(* Logix 5000 project; controller EWEB_SOCK_TCP_CLIENT_VER2_1 1756-L63 rev 15.4; software revision 15.02 *)

TASK MainTask (periodic, rate 5 ms, priority 10, watchdog 500 ms) : MainProgram

MODULES
   Local : 1756-L63 (ICP 5, rev 15.4)
END_MODULES

TYPE OpenConnParam :
STRUCT
   Timeout : DINT;
   DestAddr : STRING;
END_STRUCT
END_TYPE

TYPE READ_DATA_REQ :
STRUCT
   Timeout : DINT;
   BufLen : DINT;
END_STRUCT
END_TYPE

TYPE READ_RESP :
STRUCT
   FromAddr : SockAddr;
   READ_BUFF : STR_4096;
END_STRUCT
END_TYPE

TYPE REQUEST_PARAMETERS :
STRUCT
   Type : DINT;   // 1 - TCP 2- UPD
   Addr : SockAddr;
END_STRUCT
END_TYPE

TYPE SockAddr :
STRUCT
   Family : INT;   // Address Family Must be 2
   Port : INT;   // Port Number
   Addr : DINT;   // IP Address
END_STRUCT
END_TYPE

TYPE STR_4096 :
STRUCT
   LEN : DINT;
   DATA : SINT[4096];
END_STRUCT
END_TYPE

TYPE STR_480 :
STRUCT
   LEN : DINT;
   DATA : SINT[480];
END_STRUCT
END_TYPE

TYPE WRT_DATA :
STRUCT
   Timeout : DINT;
   ToAddr : SockAddr;
   Buffer : STR_480;
END_STRUCT
END_TYPE

VAR_GLOBAL   (* controller tags *)
   _EWEB_PATH : STRING := '$01$07';
   Accept : ALIAS FOR Log_Enable.2;
   Attrubute : ALIAS FOR Log_Enable.6;
   Buf_Len_Sent : DINT := 7;
   Change_Log_MSG : MESSAGE;
        MessageParameters(ServiceCode := 16#0010, LocalElement := Log_Enable, ...)
   CLOCK : DINT[7] := ([0] := 1998, [1] := 1, [2] := 7, [3] := 4, [4] := 26, [5] := 6, [6] := 739599);
   COLN : STRING := ':';
   Connect_MSG : MESSAGE;
        MessageParameters(ServiceCode := 16#004c, LocalElement := Sock_Open_Par, ...)
   Connect_Request : BOOL;   // Toggle This Bit to Connect to a Remote Server
   Create : ALIAS FOR Log_Enable.0;
   Create_Sock_MSG : MESSAGE;
        MessageParameters(ServiceCode := 16#004b, LocalElement := Socket, DestinationTag := Instance, ...)
   Create_Socket_Request : BOOL;   // Manually Toggle This Bit to Create Socket
   Del_All_Sockets_MSG : MESSAGE;
        MessageParameters(ServiceCode := 16#0051, ...)
   Delete : ALIAS FOR Log_Enable.5;
   Delete_All_Sockets_Request : BOOL;
   Delete_Socket_MSG : MESSAGE;
        MessageParameters(ServiceCode := 16#004f, ...)
   Delete_Socket_Request : BOOL;
   Dest_IP : STRING := '100.100.90.1';
   Dest_port : STRING := '?port=10001';
   Errors : ALIAS FOR Log_Enable.7;
   Get_Socket_Instance_MSG : MESSAGE;
        MessageParameters(ServiceCode := 16#0001, DestinationTag := Socket_Instance_DATA, ...)
   Get_Socket_Instance_Request : BOOL;
   Get_Socket_Object_MSG : MESSAGE;
        MessageParameters(ServiceCode := 16#0001, DestinationTag := Socket_Object_Class_Response, ...)
   Get_Socket_Object_Request : BOOL;
   HOUR : STRING := '4';
   Instance : DINT := 17538;
   Log_Enable : DINT;
   Log_old : DINT;
   MINUTE : STRING := '26';
   Nothing : BOOL;
   Open : ALIAS FOR Log_Enable.1;
   Read : ALIAS FOR Log_Enable.3;
   Read_Data_MSG : MESSAGE;
        MessageParameters(ServiceCode := 16#004d, LocalElement := Read_Data_Req, DestinationTag := Read_Response, ...)
   Read_Data_Req : READ_DATA_REQ := (Timeout := 1000, BufLen := 100);
   Read_Data_Request : BOOL;   // Toggle This Bit to Read Incoming TCP Data
   Read_Response : READ_RESP;
   SECOND : STRING := '06';
   Sock_Open_Par : OpenConnParam := (Timeout := 25000, DestAddr := '100.100.90.1?port=10001');
   Socket : REQUEST_PARAMETERS := (Type := 1, Addr.Family := 2, Addr.Port := 10002);
   Socket_Instance_DATA : DINT[13] := ([0] := 655491074, [4] := 2048, [5] := 2048, [6] := 8, [7] := 4, [8] := 300000);
   Socket_Object_Class_Response : SINT[10] := ([0] := 1, [2] := 20, [4] := 1);
   TIME : STRING := '4:26:06';
   Write : ALIAS FOR Log_Enable.4;
   Write_data_MSG : MESSAGE;
        MessageParameters(ServiceCode := 16#004e, LocalElement := Write_Data_Out, DestinationTag := Buf_Len_Sent, ...)
   Write_Data_Out : WRT_DATA := (Timeout := 20000, ToAddr.Family := 2, Buffer := '4:26:06');
   Write_Request : BOOL;   // Toggle This Bit to Send Data Out
   zero : STRING := '0';
END_VAR

PROGRAM MainProgram   (* main routine _SOCKET_TCP_CLIENT *)

ROUTINE _SOCKET_STATS   (* ladder *)
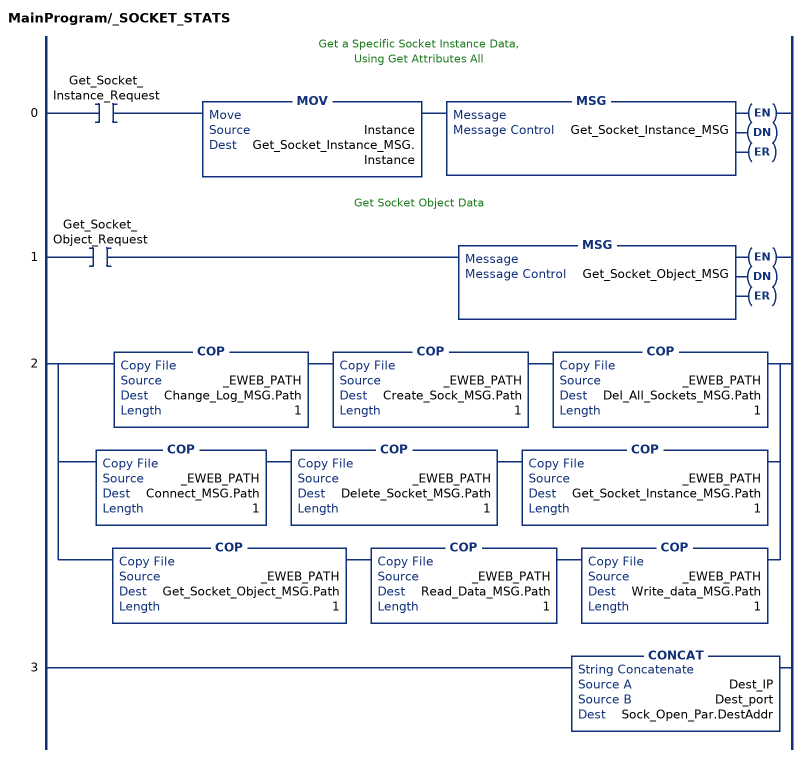
   // Get a Specific Socket Instance Data,
   // Using Get Attributes All
   0: XIC(Get_Socket_Instance_Request)MOV(Instance,Get_Socket_Instance_MSG.Instance)MSG(Get_Socket_Instance_MSG);
   // Get Socket Object Data
   1: XIC(Get_Socket_Object_Request)MSG(Get_Socket_Object_MSG);
   2: [COP(_EWEB_PATH,Change_Log_MSG.Path,1) COP(_EWEB_PATH,Create_Sock_MSG.Path,1) COP(_EWEB_PATH,Del_All_Sockets_MSG.Path,1) ,COP(_EWEB_PATH,Connect_MSG.Path,1) COP(_EWEB_PATH,Delete_Socket_MSG.Path,1) COP(_EWEB_PATH,Get_Socket_Instance_MSG.Path,1) ,COP(_EWEB_PATH,Get_Socket_Object_MSG.Path,1) COP(_EWEB_PATH,Read_Data_MSG.Path,1) COP(_EWEB_PATH,Write_data_MSG.Path,1) ];
   3: CONCAT(Dest_IP,Dest_port,Sock_Open_Par.DestAddr);
END_ROUTINE

ROUTINE _SOCKET_TCP_CLIENT   (* ladder *)
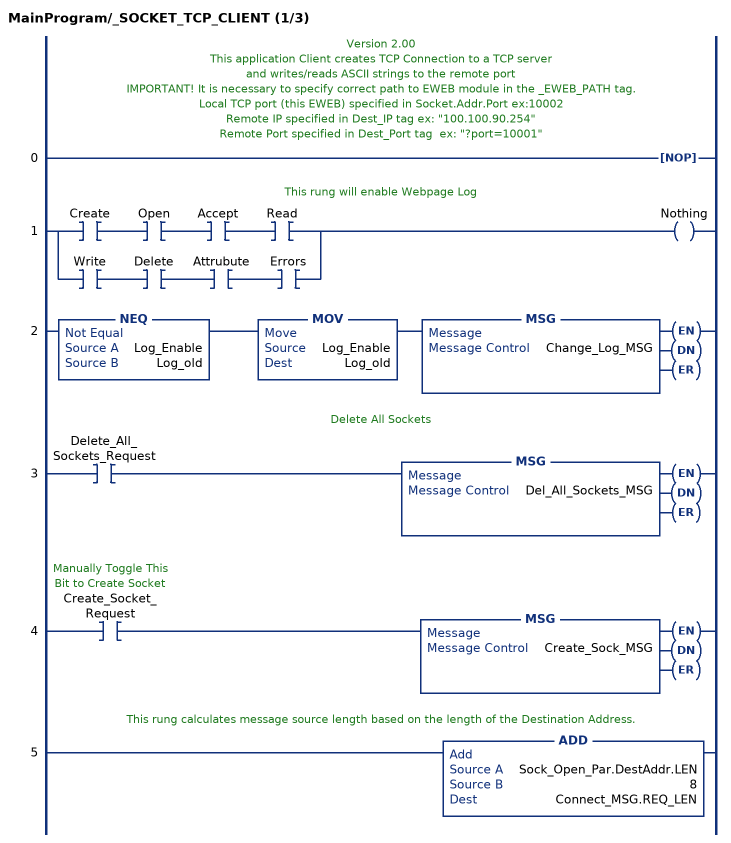
   // Version 2.00
   // This application Client creates TCP Connection to a TCP server
   // and writes/reads ASCII strings to the remote port
   // IMPORTANT! It is necessary to specify correct path to EWEB module in the _EWEB_PATH tag.
   // Local TCP port (this EWEB) specified in Socket.Addr.Port ex:10002
   // Remote IP specified in Dest_IP tag ex: "100.100.90.254"
   // Remote Port specified in Dest_Port tag  ex: "?port=10001"
   0: NOP();
   // This rung will enable Webpage Log
   1: [XIC(Create) XIC(Open) XIC(Accept) XIC(Read) ,XIC(Write) XIC(Delete) XIC(Attrubute) XIC(Errors) ]OTE(Nothing);
   2: NEQ(Log_Enable,Log_old)MOV(Log_Enable,Log_old)MSG(Change_Log_MSG);
   // Delete All Sockets
   3: XIC(Delete_All_Sockets_Request)MSG(Del_All_Sockets_MSG);
   4: XIC(Create_Socket_Request)MSG(Create_Sock_MSG);
   // This rung calculates message source length based on the length of the Destination Address.
   5: ADD(Sock_Open_Par.DestAddr.LEN,8,Connect_MSG.REQ_LEN);
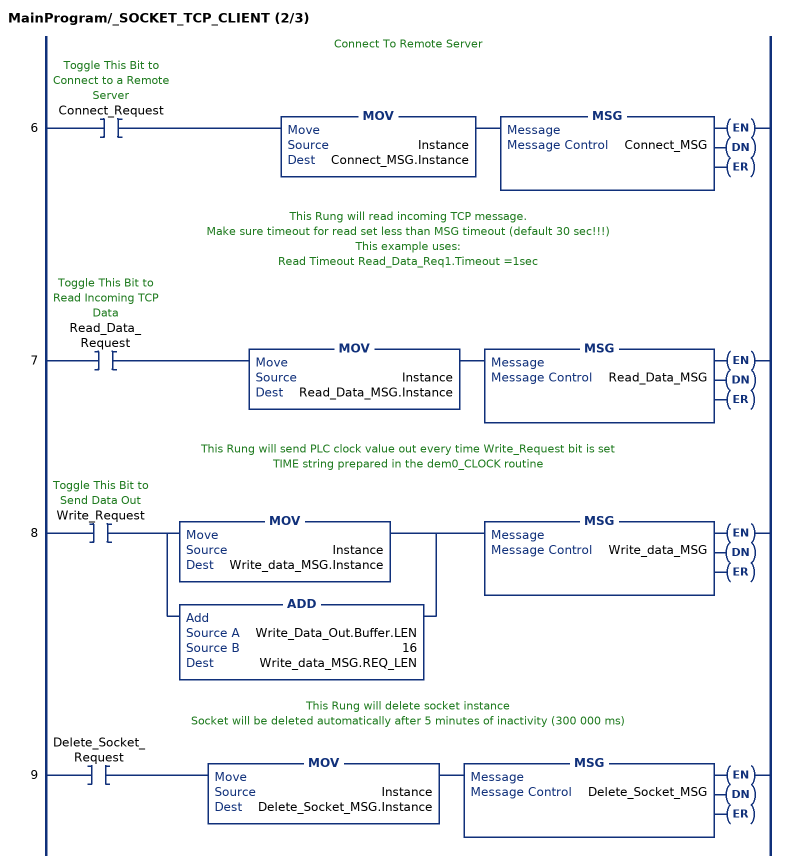
   // Connect To Remote Server
   6: XIC(Connect_Request)MOV(Instance,Connect_MSG.Instance)MSG(Connect_MSG);
   // This Rung will read incoming TCP message.
   // Make sure timeout for read set less than MSG timeout (default 30 sec!!!)
   // This example uses:
   // Read Timeout Read_Data_Req1.Timeout =1sec
   7: XIC(Read_Data_Request)MOV(Instance,Read_Data_MSG.Instance)MSG(Read_Data_MSG);
   // This Rung will send PLC clock value out every time Write_Request bit is set
   // TIME string prepared in the dem0_CLOCK routine
   8: XIC(Write_Request)[MOV(Instance,Write_data_MSG.Instance) ,ADD(Write_Data_Out.Buffer.LEN,16,Write_data_MSG.REQ_LEN) ]MSG(Write_data_MSG);
   // This Rung will delete socket instance
   // Socket will be deleted automatically after 5 minutes of inactivity (300 000 ms)
   9: XIC(Delete_Socket_Request)MOV(Instance,Delete_Socket_MSG.Instance)MSG(Delete_Socket_MSG);
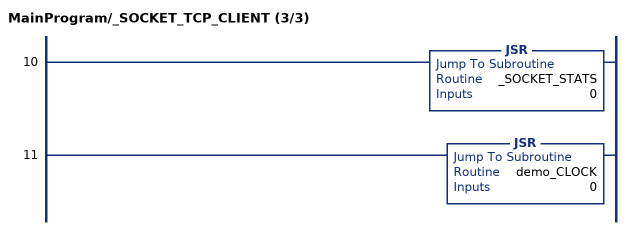
   10: JSR(_SOCKET_STATS,0);
   11: JSR(demo_CLOCK,0);
END_ROUTINE

ROUTINE demo_CLOCK   (* ladder *)
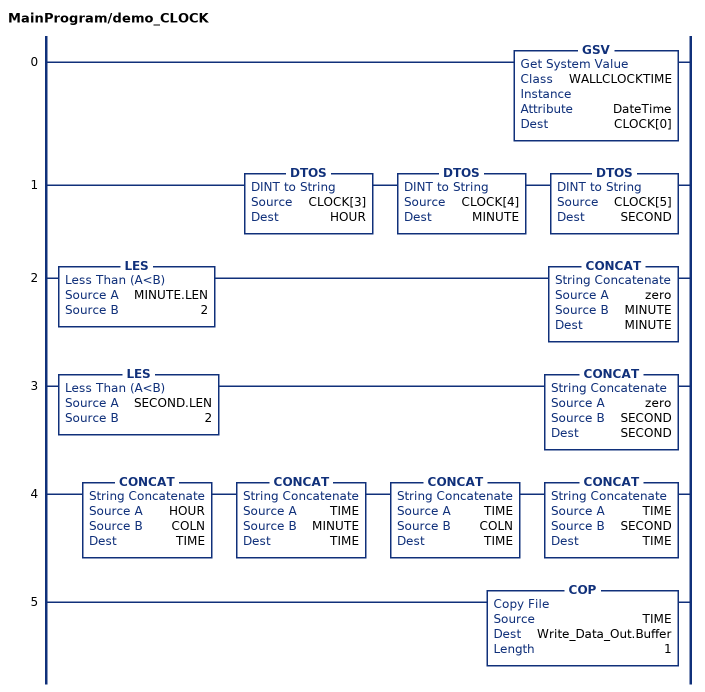
   0: GSV(WALLCLOCKTIME,,DateTime,CLOCK[0]);
   1: DTOS(CLOCK[3],HOUR)DTOS(CLOCK[4],MINUTE)DTOS(CLOCK[5],SECOND);
   2: LES(MINUTE.LEN,2)CONCAT(zero,MINUTE,MINUTE);
   3: LES(SECOND.LEN,2)CONCAT(zero,SECOND,SECOND);
   4: CONCAT(HOUR,COLN,TIME)CONCAT(TIME,MINUTE,TIME)CONCAT(TIME,COLN,TIME)CONCAT(TIME,SECOND,TIME);
   5: COP(TIME,Write_Data_Out.Buffer,1);
END_ROUTINE
END_PROGRAM
